// TIA Portal V20 export
DATA_BLOCK "T10 LANT HMI"   // DB1293
{ S7_Optimized_Access := 'TRUE' }
AUTHOR : SAS
// stored: AutoNumber false, IsRetainMemResEnabled true, MemoryReserve 100, RetainMemoryReserve 100
   VAR
      Conditions : Struct
         CG : "Pop_Up_Aux";   // General conditions
         CA : "Pop_Up_Aux";   // Start Auto mode conditions
         SC : "Pop_Up_Aux";   // Start cycle conditions
         MOV_FW : "Pop_Up_Aux";   // Movement interlocks Forward
         MOV_BW : "Pop_Up_Aux";   // Movement interlocks Backward
      END_STRUCT;
      HMI : Struct
         PB : Struct
            s0 : Bool;
            s1 : Bool;
            s2 : Bool;
            s3 : Bool;
            s4 : Bool;
            Pause : Bool;   // Pause
            s6 : Bool;
            s7 : Bool;
            s8 : Bool;
            s9 : Bool;
            s10 : Bool;
            s11 : Bool;
            s12 : Bool;
            s13 : Bool;
            s14 : Bool;
            s15 : Bool;
         END_STRUCT;
         ST : Struct
            s0 : Bool;
            s1 : Bool;
            s2 : Bool;
            s3 : Bool;
            s4 : Bool;
            Pause : Bool;   // Pause
            s6 : Bool;
            s7 : Bool;
            s8 : Bool;
            s9 : Bool;
            "ST Machine" : Int;   // Device label status (0=EME, 1=Safe, 2=Fault, 3=Run, 4=Stopped)
            "ST Sequencer step" : Int;   // Sequencer step
         END_STRUCT;
      END_STRUCT;
   END_VAR
BEGIN
   // Conditions.CG.Conditions.n1 : Tensiune Alimentare OK
   // Conditions.CG.Conditions.n2 : Electric protectie OK
   // Conditions.CG.Conditions.n3 : Inverter OK
   // Conditions.CA.Conditions.n1 : Conditiie Generale
   // Conditions.SC.Conditions.n1 : Initial Conditions
   // Conditions.SC.Conditions.n2 : Piece Presence
   // Conditions.SC.Conditions.n3 : Tracking OK
   // Conditions.SC.Conditions.n4 : Condition of movement
   // Conditions.SC.Conditions.n5 : Excentric Stopped
   // Conditions.SC.Conditions.n6 : Opritor Pozitie Sus
   // Conditions.MOV_FW.Conditions.n1 : Permanent Conditions
   // Conditions.MOV_BW.Conditions.n1 : Permanent Conditions
END_DATA_BLOCK
